PROGRAM POU_Lights
VAR_INPUT
bAxesEnablem:BOOL;
bEStop:BOOL;
END_VAR
VAR
tTimeLightOn:TIME:=T#0S;
tTimeStartMove:TIME;
tCurrentLight:TIME;
tCurrentMoveDur:TIME;
bLightRed  AT%Q* : BOOL;
bLightAmber  AT%Q* : BOOL;
bLightGreen  AT%Q* : BOOL;
END_VAR

IF bEStop AND bLimits AND bMotorError
	THEN
	

IF bAxis1Enable OR bAxis2Enable OR bAxis3Enable OR bAxis4Enable OR bAxis5Enable OR bAxis6Enable
	
	THEN
	tCurrentLight:=TIME();
	tCurrentMoveDur:=tCurrentLight-tTimeLightOn;
	IF (tCurrentMoveDur < T#1S)  
		THEN
		bLightRed:=FALSE;
		bLightAmber:=TRUE;
		bLightGreen:=FALSE;
	END_IF
	IF (tCurrentMoveDur > T#1S)AND (tCurrentMoveDur < T#2S)
		THEN
		bLightRed:=FALSE;
		bLightAmber:=FALSE;
		bLightGreen:=FALSE;
	END_IF
	IF (tCurrentMoveDur > T#2S)
		THEN
		tTimeLightOn:=TIME();
	END_IF
	ELSE
	tTimeLightOn:=TIME();	
	bLightRed:=FALSE;
	bLightAmber:=FALSE;
	bLightGreen:=TRUE;
END_IF
ELSE
	bLightRed:=TRUE;
	bLightAmber:=FALSE;
	bLightGreen:=FALSE;
END_IF

END_PROGRAM

(* stored: Version 1.1.0.1, ProductVersion 3.1.4022.18
   POU POU_Lights: Id {2cc51798-d30b-4ad9-813c-6d16cd0fcc10}, SpecialFunc None *)
